PROGRAM PRG_RotDet
VAR
    fb_Rot_Det : FB_MotionStage;
    bInit : BOOl := TRUE;
END_VAR

IF ( bInit) THEN
   bInit := FALSE;
   Main.M45.bHardwareEnable := TRUE;
   Main.M45.bPowerSelf := TRUE;
   Main.M45.nBrakeMode := ENUM_StageBrakeMode.NO_BRAKE;
   Main.M45.nEnableMode := ENUM_StageEnableMode.DURING_MOTION;
   Main.M45.bLimitForwardEnable := TRUE;
   Main.M45.bLimitBackwardEnable := TRUE;
END_IF

fb_Rot_Det(stMotionStage:=Main.M45);

END_PROGRAM

(* stored: Version 1.1.0.1, ProductVersion 3.1.4024.12
   POU PRG_RotDet: Id {6c5a9ec6-70ef-4f3f-9260-ca012a2c65e6}, SpecialFunc None *)
